{attribute addProperty BoxType "EL1262-0000-0002"}
{attribute addProperty Id "Ch1_CycleCountAT %I*UINT162"}
{attribute addProperty CRC "790658108"}
{attribute addProperty SizeInBites "16"}
{attribute addProperty SizeInBytes "2"}
TYPE Ch1_CycleCount_2F207C3C :
STRUCT
	{attribute addProperty Name "Ch1_CycleCount"}
	Ch1_CycleCount AT %I* : UINT;
END_STRUCT
END_TYPE

(* stored: Version 1.2.0.0, ProductVersion 3.1.4024.9
   DUT Ch1_CycleCount_2F207C3C: Id {06be53de-79b7-4740-bb2b-9bdb2cc200da} *)
